// TIA Portal V20 export
FUNCTION_BLOCK "FB_HMI"   // FB11, LAD
{ S7_Optimized_Access := 'TRUE' }
// stored: AutoNumber false, MemoryReserve 100, SetENOAutomatically false
   VAR_INPUT
      Control_Screen_HMI : Word;
      Employee_Rework : String[6];
      Admin_1 : String[6] := '';
      Admin_2 : String[6];
      Admin_3 : String[6];
      Admin_4 : String[6];
      Admin_5 : String[6];
      Alarm_0 : Word;
      Alarm_1 : Word;
      Alarm_2 : Word;
   END_VAR
   VAR_OUTPUT
      Alarm : Bool;
      Job_Mailbox : Array[0..3] of Word;
   END_VAR
   VAR
      Aux_Trigger_0 : Bool;
      Aux_Trigger_1 : Bool;
      Aux_Trigger_2 : Bool;
      Aux_Trigger_3 : Bool;
      Aux_Trigger_4 : Bool;
      Aux_Trigger_5 : Bool;
      Aux_Trigger_6 : Bool;
      Aux_Trigger_7 : Bool;
      Aux_Trigger_8 : Bool;
      Aux_Trigger_9 : Bool;
      Aux_Trigger_10 : Bool;
      Everybody_Can_Access : Bool;
      Only_Admin_Can_Access : Bool;
      Control_Screen : Word;
      Timer_Delay_Change_Screen { S7_SetPoint := 'True'} : TON_TIME;
      Timer_Delay_Change_Job_Mailbox { S7_SetPoint := 'True'} : TON_TIME;
   END_VAR
   VAR CONSTANT
      Screen_1 : Word := 16#1;
      Screen_2 : Word := 16#2;
      Screen_3 : Word := 16#3;
      Screen_4 : Word := 16#4;
      Screen_5 : Word := 16#5;
      Screen_6 : Word := 16#6;
      Screen_7 : Word := 16#7;
      Screen_8 : Word := 16#8;
      Screen_9 : Word := 16#9;
      Screen_10 : Word := 16#20;
      Screen_11 : Word := 16#21;
      Screen_12 : Word := 16#22;
      Screen_13 : Word := 16#23;
      Screen_14 : Word := 16#24;
      Lau : String := 'Lau$R$00$00';
   END_VAR
   // Job_Mailbox[0] := 51;
   // Job_Mailbox[2..3] := 0;
   VAR_TEMP   // added for the SCL form of the ladder/FBD networks
      _w1 : Bool;
      _w2 : Bool;
      _w3 : Bool;
   END_VAR
BEGIN

REGION Network 1: Admin
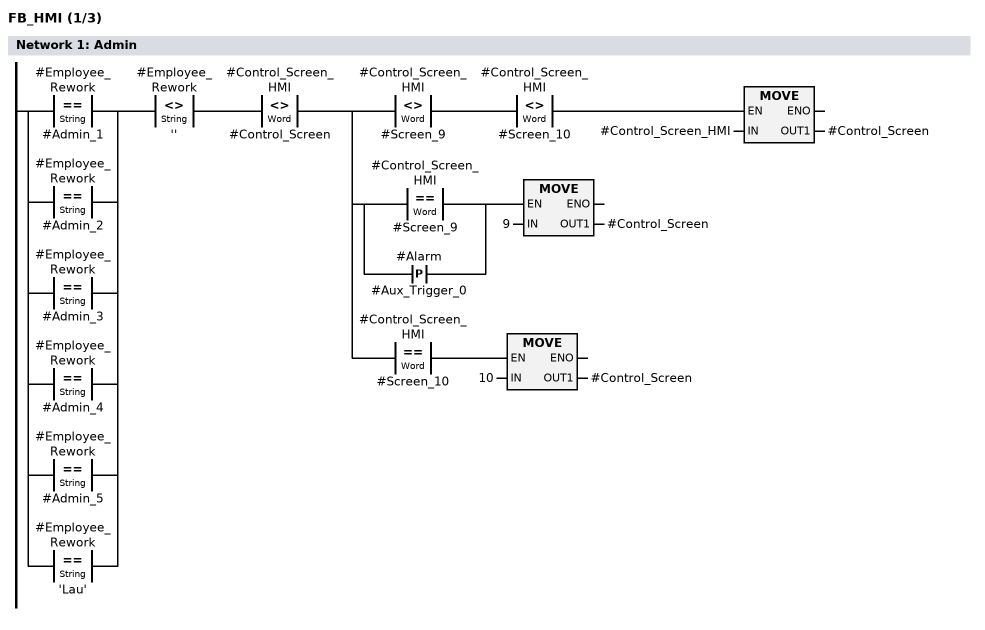
   RUNG wire#powerrail
      { S7_Templates := "SrcType := String" } EQ_Contact(in1 := #Employee_Rework, in2 := #Admin_1)
      wire#w1
      { S7_Templates := "SrcType := String" } NE_Contact(in1 := #Employee_Rework, in2 := '')
      { S7_Templates := "SrcType := Word" } NE_Contact(in1 := #Control_Screen_HMI, in2 := #Control_Screen)
      wire#w2
      { S7_Templates := "SrcType := Word" } NE_Contact(in1 := #Control_Screen_HMI, in2 := #Screen_9)
      { S7_Templates := "SrcType := Word" } NE_Contact(in1 := #Control_Screen_HMI, in2 := #Screen_10)
      Move(in := #Control_Screen_HMI, out1 => #Control_Screen)
   END_RUNG
   RUNG wire#powerrail
      { S7_Templates := "SrcType := String" } EQ_Contact(in1 := #Employee_Rework, in2 := #Admin_2)
   END_RUNG wire#w1
   RUNG wire#powerrail
      { S7_Templates := "SrcType := String" } EQ_Contact(in1 := #Employee_Rework, in2 := #Admin_3)
   END_RUNG wire#w1
   RUNG wire#powerrail
      { S7_Templates := "SrcType := String" } EQ_Contact(in1 := #Employee_Rework, in2 := #Admin_4)
   END_RUNG wire#w1
   RUNG wire#powerrail
      { S7_Templates := "SrcType := String" } EQ_Contact(in1 := #Employee_Rework, in2 := #Admin_5)
   END_RUNG wire#w1
   RUNG wire#powerrail
      { S7_Templates := "SrcType := String" } EQ_Contact(in1 := #Employee_Rework, in2 := 'Lau')
   END_RUNG wire#w1
   RUNG wire#w2
      { S7_Templates := "SrcType := Word" } EQ_Contact(in1 := #Control_Screen_HMI, in2 := #Screen_9)
      wire#w3
      Move(in := 9, out1 => #Control_Screen)
   END_RUNG
   RUNG wire#w2
      P_Contact(operand := #Alarm, bit := #Aux_Trigger_0)
   END_RUNG wire#w3
   RUNG wire#w2
      { S7_Templates := "SrcType := Word" } EQ_Contact(in1 := #Control_Screen_HMI, in2 := #Screen_10)
      Move(in := 10, out1 => #Control_Screen)
   END_RUNG
   // the same network as SCL:
   #_w1 := ((#Employee_Rework = #Admin_1) OR (#Employee_Rework = #Admin_2) OR (#Employee_Rework = #Admin_3) OR (#Employee_Rework = #Admin_4) OR (#Employee_Rework = #Admin_5) OR (#Employee_Rework = 'Lau')) AND (#Employee_Rework <> '') AND (#Control_Screen_HMI <> #Control_Screen);
   IF #_w1 AND (#Control_Screen_HMI <> #Screen_9) AND (#Control_Screen_HMI <> #Screen_10) THEN
       #Control_Screen := #Control_Screen_HMI;
   END_IF;
   #_w2 := #_w1 AND #Alarm AND NOT #Aux_Trigger_0;   // rising edge of #Alarm
   #Aux_Trigger_0 := #Alarm;
   IF (#_w1 AND (#Control_Screen_HMI = #Screen_9)) OR #_w2 THEN #Control_Screen := 9; END_IF;
   IF #_w1 AND (#Control_Screen_HMI = #Screen_10) THEN #Control_Screen := 10; END_IF;
END_REGION

REGION Network 2
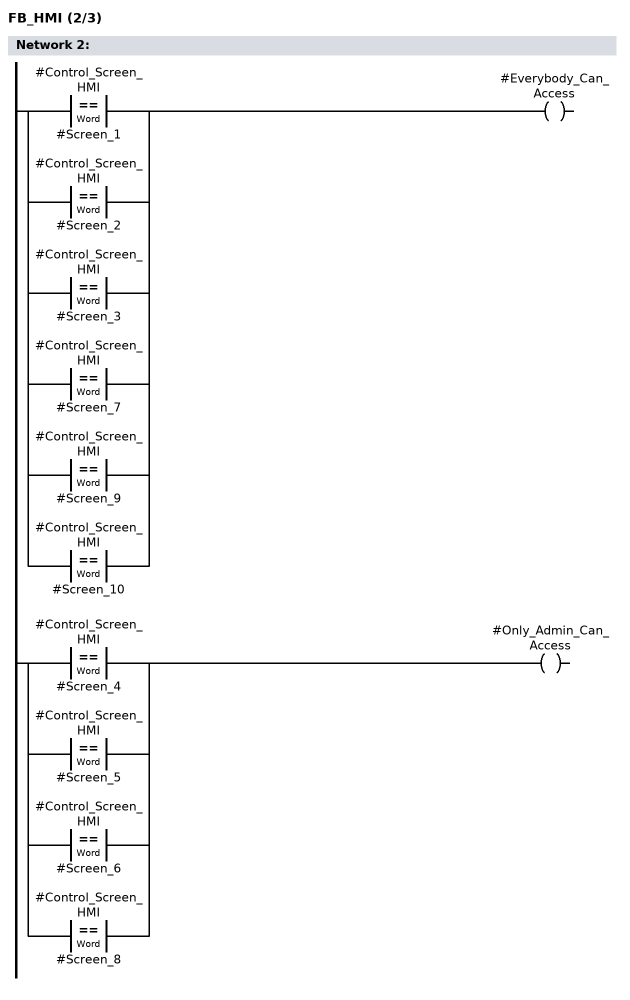
   RUNG wire#powerrail
      { S7_Templates := "SrcType := Word" } EQ_Contact(in1 := #Control_Screen_HMI, in2 := #Screen_1)
      wire#w1
      Coil( #Everybody_Can_Access )
   END_RUNG
   RUNG wire#powerrail
      { S7_Templates := "SrcType := Word" } EQ_Contact(in1 := #Control_Screen_HMI, in2 := #Screen_2)
   END_RUNG wire#w1
   RUNG wire#powerrail
      { S7_Templates := "SrcType := Word" } EQ_Contact(in1 := #Control_Screen_HMI, in2 := #Screen_3)
   END_RUNG wire#w1
   RUNG wire#powerrail
      { S7_Templates := "SrcType := Word" } EQ_Contact(in1 := #Control_Screen_HMI, in2 := #Screen_7)
   END_RUNG wire#w1
   RUNG wire#powerrail
      { S7_Templates := "SrcType := Word" } EQ_Contact(in1 := #Control_Screen_HMI, in2 := #Screen_9)
   END_RUNG wire#w1
   RUNG wire#powerrail
      { S7_Templates := "SrcType := Word" } EQ_Contact(in1 := #Control_Screen_HMI, in2 := #Screen_10)
   END_RUNG wire#w1
   RUNG wire#powerrail
      { S7_Templates := "SrcType := Word" } EQ_Contact(in1 := #Control_Screen_HMI, in2 := #Screen_4)
      wire#w2
      Coil( #Only_Admin_Can_Access )
   END_RUNG
   RUNG wire#powerrail
      { S7_Templates := "SrcType := Word" } EQ_Contact(in1 := #Control_Screen_HMI, in2 := #Screen_5)
   END_RUNG wire#w2
   RUNG wire#powerrail
      { S7_Templates := "SrcType := Word" } EQ_Contact(in1 := #Control_Screen_HMI, in2 := #Screen_6)
   END_RUNG wire#w2
   RUNG wire#powerrail
      { S7_Templates := "SrcType := Word" } EQ_Contact(in1 := #Control_Screen_HMI, in2 := #Screen_8)
   END_RUNG wire#w2
   // the same network as SCL:
   #Everybody_Can_Access := (#Control_Screen_HMI = #Screen_1) OR (#Control_Screen_HMI = #Screen_2) OR (#Control_Screen_HMI = #Screen_3) OR (#Control_Screen_HMI = #Screen_7) OR (#Control_Screen_HMI = #Screen_9) OR (#Control_Screen_HMI = #Screen_10);
   #Only_Admin_Can_Access := (#Control_Screen_HMI = #Screen_4) OR (#Control_Screen_HMI = #Screen_5) OR (#Control_Screen_HMI = #Screen_6) OR (#Control_Screen_HMI = #Screen_8);
END_REGION

REGION Network 3: Not Admin
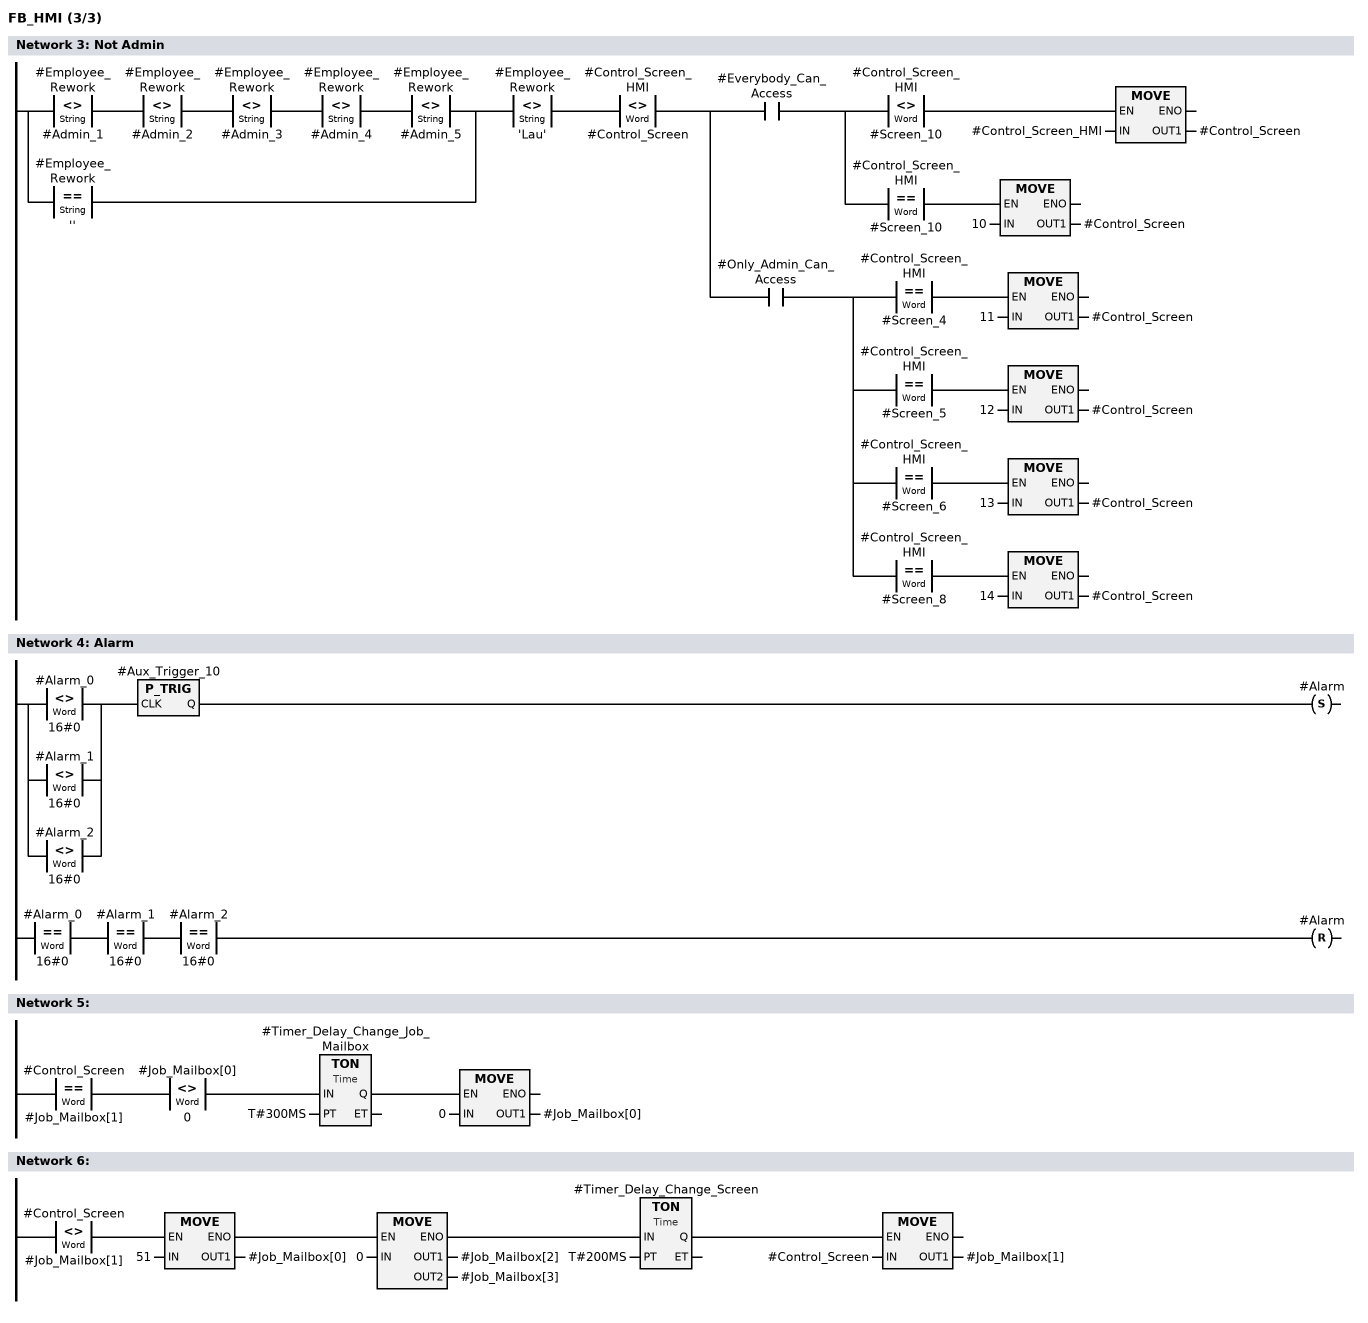
   RUNG wire#powerrail
      { S7_Templates := "SrcType := String" } NE_Contact(in1 := #Employee_Rework, in2 := #Admin_1)
      { S7_Templates := "SrcType := String" } NE_Contact(in1 := #Employee_Rework, in2 := #Admin_2)
      { S7_Templates := "SrcType := String" } NE_Contact(in1 := #Employee_Rework, in2 := #Admin_3)
      { S7_Templates := "SrcType := String" } NE_Contact(in1 := #Employee_Rework, in2 := #Admin_4)
      { S7_Templates := "SrcType := String" } NE_Contact(in1 := #Employee_Rework, in2 := #Admin_5)
      wire#w1
      { S7_Templates := "SrcType := String" } NE_Contact(in1 := #Employee_Rework, in2 := 'Lau')
      { S7_Templates := "SrcType := Word" } NE_Contact(in1 := #Control_Screen_HMI, in2 := #Control_Screen)
      wire#w2
      Contact( #Everybody_Can_Access )
      wire#w3
      { S7_Templates := "SrcType := Word" } NE_Contact(in1 := #Control_Screen_HMI, in2 := #Screen_10)
      Move(in := #Control_Screen_HMI, out1 => #Control_Screen)
   END_RUNG
   RUNG wire#powerrail
      { S7_Templates := "SrcType := String" } EQ_Contact(in1 := #Employee_Rework, in2 := '')
   END_RUNG wire#w1
   RUNG wire#w3
      { S7_Templates := "SrcType := Word" } EQ_Contact(in1 := #Control_Screen_HMI, in2 := #Screen_10)
      Move(in := 10, out1 => #Control_Screen)
   END_RUNG
   RUNG wire#w2
      Contact( #Only_Admin_Can_Access )
      wire#w4
      { S7_Templates := "SrcType := Word" } EQ_Contact(in1 := #Control_Screen_HMI, in2 := #Screen_4)
      Move(in := 11, out1 => #Control_Screen)
   END_RUNG
   RUNG wire#w4
      { S7_Templates := "SrcType := Word" } EQ_Contact(in1 := #Control_Screen_HMI, in2 := #Screen_5)
      Move(in := 12, out1 => #Control_Screen)
   END_RUNG
   RUNG wire#w4
      { S7_Templates := "SrcType := Word" } EQ_Contact(in1 := #Control_Screen_HMI, in2 := #Screen_6)
      Move(in := 13, out1 => #Control_Screen)
   END_RUNG
   RUNG wire#w4
      { S7_Templates := "SrcType := Word" } EQ_Contact(in1 := #Control_Screen_HMI, in2 := #Screen_8)
      Move(in := 14, out1 => #Control_Screen)
   END_RUNG
   // the same network as SCL:
   #_w1 := (((#Employee_Rework <> #Admin_1) AND (#Employee_Rework <> #Admin_2) AND (#Employee_Rework <> #Admin_3) AND (#Employee_Rework <> #Admin_4) AND (#Employee_Rework <> #Admin_5)) OR (#Employee_Rework = '')) AND (#Employee_Rework <> 'Lau') AND (#Control_Screen_HMI <> #Control_Screen);
   #_w2 := #_w1 AND #Everybody_Can_Access;
   IF #_w2 AND (#Control_Screen_HMI <> #Screen_10) THEN #Control_Screen := #Control_Screen_HMI; END_IF;
   IF #_w2 AND (#Control_Screen_HMI = #Screen_10) THEN #Control_Screen := 10; END_IF;
   #_w3 := #_w1 AND #Only_Admin_Can_Access;
   IF #_w3 AND (#Control_Screen_HMI = #Screen_4) THEN #Control_Screen := 11; END_IF;
   IF #_w3 AND (#Control_Screen_HMI = #Screen_5) THEN #Control_Screen := 12; END_IF;
   IF #_w3 AND (#Control_Screen_HMI = #Screen_6) THEN #Control_Screen := 13; END_IF;
   IF #_w3 AND (#Control_Screen_HMI = #Screen_8) THEN #Control_Screen := 14; END_IF;
END_REGION

REGION Network 4: Alarm
   RUNG wire#powerrail
      { S7_Templates := "SrcType := Word" } NE_Contact(in1 := #Alarm_0, in2 := 16#0)
      wire#w1
      P_Trig( #Aux_Trigger_10 )
      S_Coil( #Alarm )
   END_RUNG
   RUNG wire#powerrail
      { S7_Templates := "SrcType := Word" } NE_Contact(in1 := #Alarm_1, in2 := 16#0)
   END_RUNG wire#w1
   RUNG wire#powerrail
      { S7_Templates := "SrcType := Word" } NE_Contact(in1 := #Alarm_2, in2 := 16#0)
   END_RUNG wire#w1
   RUNG wire#powerrail
      { S7_Templates := "SrcType := Word" } EQ_Contact(in1 := #Alarm_0, in2 := 16#0)
      { S7_Templates := "SrcType := Word" } EQ_Contact(in1 := #Alarm_1, in2 := 16#0)
      { S7_Templates := "SrcType := Word" } EQ_Contact(in1 := #Alarm_2, in2 := 16#0)
      R_Coil( #Alarm )
   END_RUNG
   // the same network as SCL:
   #_w1 := (#Alarm_0 <> 16#0) OR (#Alarm_1 <> 16#0) OR (#Alarm_2 <> 16#0);
   #_w2 := #_w1 AND NOT #Aux_Trigger_10;   // rising edge
   #Aux_Trigger_10 := #_w1;
   IF #_w2 THEN #Alarm := TRUE; END_IF;
   IF (#Alarm_0 = 16#0) AND (#Alarm_1 = 16#0) AND (#Alarm_2 = 16#0) THEN #Alarm := FALSE; END_IF;
END_REGION

REGION Network 5
   RUNG wire#powerrail
      { S7_Templates := "SrcType := Word" } EQ_Contact(in1 := #Control_Screen, in2 := #Job_Mailbox[1])
      { S7_Templates := "SrcType := Word" } NE_Contact(in1 := #Job_Mailbox[0], in2 := 0)
      { S7_Templates := "time_type := Time" } #Timer_Delay_Change_Job_Mailbox.TON(pt := T#300MS, et =>)
      Move(in := 0, out1 => #Job_Mailbox[0])
   END_RUNG
   // the same network as SCL:
   #Timer_Delay_Change_Job_Mailbox(IN := (#Control_Screen = #Job_Mailbox[1]) AND (#Job_Mailbox[0] <> 0),   // TON
                           PT := T#300MS);
   IF #Timer_Delay_Change_Job_Mailbox.Q THEN #Job_Mailbox[0] := 0; END_IF;
END_REGION

REGION Network 6
   RUNG wire#powerrail
      { S7_Templates := "SrcType := Word" } NE_Contact(in1 := #Control_Screen, in2 := #Job_Mailbox[1])
      Move(in := 51, out1 => #Job_Mailbox[0])
      Move(in := 0, out1 => #Job_Mailbox[2], out2 => #Job_Mailbox[3])
      { S7_Templates := "time_type := Time" } #Timer_Delay_Change_Screen.TON(pt := T#200MS, et =>)
      Move(in := #Control_Screen, out1 => #Job_Mailbox[1])
   END_RUNG
   // the same network as SCL:
   #_w1 := #Control_Screen <> #Job_Mailbox[1];
   IF #_w1 THEN
       #Job_Mailbox[0] := 51;
       #Job_Mailbox[2] := 0;
       #Job_Mailbox[3] := 0;
   END_IF;
   #Timer_Delay_Change_Screen(IN := #_w1, PT := T#200MS);   // TON
   IF #Timer_Delay_Change_Screen.Q THEN #Job_Mailbox[1] := #Control_Screen; END_IF;
END_REGION
END_FUNCTION_BLOCK
